// TIA Portal V21 export
VAR_GLOBAL   // PLC tag table "KAllValvola"
END_VAR
VAR_GLOBAL CONSTANT   // user constants
   KAllValv_TimeOutPosiz : Int := 1;   // Timeout Ventilpositionierung / Valve positioning timeout / Timeout posicionamiento válvula / Délai de positionnement de la vanne / Timeout posizionamento valvola
   KAllValv_ValvolaNonInAuto : Int := 2;   // Ventil nicht in Automatik / Valve not in automatic mode / Válvula no en automático / Vanne non automatique / Valvola non in automatico
   KAllValv_ResetRichiesto : Int := 3;   // Zurücksetzen erforderlich / Reset request / Reset requerido / Réinitialisation requise / Reset richiesto
   KAllValv_ByPassFinecorsa : Int := 4;   // Bypass Endschalter / Limit switch bypass / Bypass final de carrera / Bypass de fin de course / Bypass finecorsa
END_VAR
